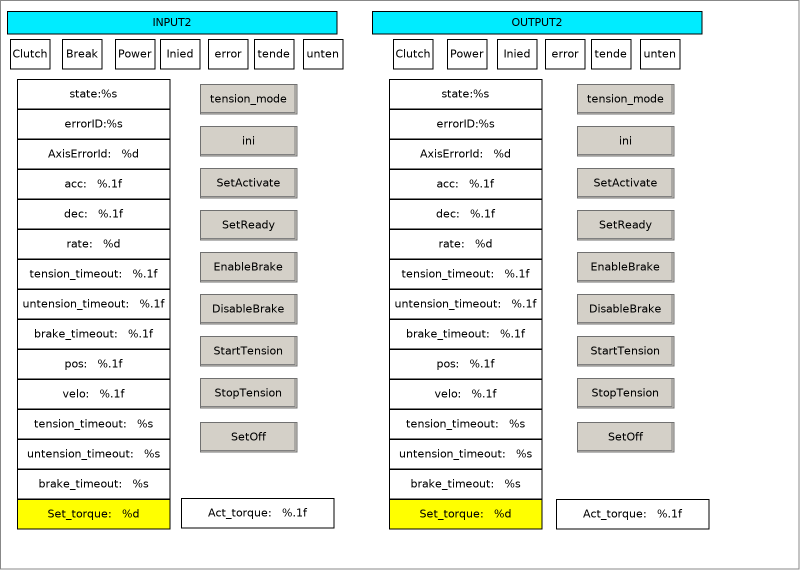
VISUALIZATION VIS_RTR_2  // 800x570
    RoundedRectangle (372,11 330x23), "OUTPUT2"
    RoundedRectangle (7,11 330x23), "INPUT2"
    Rectangle (17,79 153x30), "state:%s", colour toggle: GVL_API.stRoolToRool[3].state=100, text list: 'TextList_RTRstate', text index: GVL_API.stRoolToRool[3].state
    Rectangle (17,109 153x30), "errorID:%s", colour toggle: GVL_API.stRoolToRool[3].error_code<>0, text list: 'TextList_RTR_errorid', text index: GVL_API.stRoolToRool[3].error_code
    Rectangle (17,169 153x30), "acc: %.1f", text variable: GVL_API.stRoolToRool[3].acceleration
        OnMouseDown: write GVL_API.stRoolToRool[3].acceleration via Default
    Rectangle (17,199 153x30), "dec: %.1f", text variable: GVL_API.stRoolToRool[3].deceleration
        OnMouseDown: write GVL_API.stRoolToRool[3].deceleration via Default
    Rectangle (17,229 153x30), "rate: %d", text variable: GVL_API.stRoolToRool[3].rate
        OnMouseDown: write GVL_API.stRoolToRool[3].rate via Default
    Rectangle (17,259 153x30), "tension_timeout: %.1f", text variable: GVL_API.stRoolToRool[3].tension_timeout
        OnMouseDown: write GVL_API.stRoolToRool[3].tension_timeout via Default
    Rectangle (17,289 153x30), "untension_timeout: %.1f", text variable: GVL_API.stRoolToRool[3].untension_timeout
        OnMouseDown: write GVL_API.stRoolToRool[3].untension_timeout via Default
    Rectangle (17,319 153x30), "brake_timeout: %.1f", text variable: GVL_API.stRoolToRool[3].brake_timeout
        OnMouseDown: write GVL_API.stRoolToRool[3].brake_timeout via Default
    Rectangle (17,139 153x30), "AxisErrorId: %d", text variable: GVL_API.stRoolToRool[3].AxisErrorId
    RoundedRectangle (10,39 40x30), "Clutch", colour toggle: stOutput .bqCluthOut[3]
    RoundedRectangle (62,39 40x30), "Break", colour toggle: stOutput.bqBreakPower[3]
    Rectangle (389,79 153x30), "state:%s", colour toggle: GVL_API.stRoolToRool[4].state=100, text list: 'TextList_RTRstate', text index: GVL_API.stRoolToRool[4].state
    Rectangle (389,109 153x30), "errorID:%s", colour toggle: GVL_API.stRoolToRool[3].error_code<>0, text list: 'TextList_RTR_errorid', text index: GVL_API.stRoolToRool[4].error_code
    Rectangle (389,169 153x30), "acc: %.1f", text variable: GVL_API.stRoolToRool[4].acceleration
        OnMouseDown: write GVL_API.stRoolToRool[4].acceleration via Default
    Rectangle (389,199 153x30), "dec: %.1f", text variable: GVL_API.stRoolToRool[4].deceleration
        OnMouseDown: write GVL_API.stRoolToRool[4].deceleration via Default
    Rectangle (389,229 153x30), "rate: %d", text variable: GVL_API.stRoolToRool[4].rate
        OnMouseDown: write GVL_API.stRoolToRool[4].rate via Default
    Rectangle (389,259 153x30), "tension_timeout: %.1f", text variable: GVL_API.stRoolToRool[4].tension_timeout
        OnMouseDown: write GVL_API.stRoolToRool[4].tension_timeout via Default
    Rectangle (389,289 153x30), "untension_timeout: %.1f", text variable: GVL_API.stRoolToRool[4].untension_timeout
        OnMouseDown: write GVL_API.stRoolToRool[4].untension_timeout via Default
    Rectangle (389,319 153x30), "brake_timeout: %.1f", text variable: GVL_API.stRoolToRool[4].brake_timeout
        OnMouseDown: write GVL_API.stRoolToRool[4].brake_timeout via Default
    Rectangle (389,139 153x30), "AxisErrorId: %d", text variable: GVL_API.stRoolToRool[4].AxisErrorId
    RoundedRectangle (393,39 40x30), "Clutch", colour toggle: stOutput .bqCluthOut[4]
    Button (200,126 97x30), "ini", colour toggle: GVL_API.stRoolToRool[3].Initialize
        toggle GVL_API.stRoolToRool[3].Initialize
    Button (200,84 97x30), "tension_mode", colour toggle: GVL_API.stRoolToRool[3].tension_mode
        toggle GVL_API.stRoolToRool[3].tension_mode
    Button (200,168 97x30), "SetActivate", colour toggle: GVL_API.stRoolToRool[3].SetActivate
        toggle GVL_API.stRoolToRool[3].SetActivate
    Button (200,294 97x30), "DisableBrake", colour toggle: GVL_API.stRoolToRool[3].DisableBrake
        toggle GVL_API.stRoolToRool[3].DisableBrake
    Button (200,210 97x30), "SetReady", colour toggle: GVL_API.stRoolToRool[3].SetReady
        toggle GVL_API.stRoolToRool[3].SetReady
    Button (200,252 97x30), "EnableBrake", colour toggle: GVL_API.stRoolToRool[3].EnableBrake
        toggle GVL_API.stRoolToRool[3].EnableBrake
    Button (200,336 97x30), "StartTension", colour toggle: GVL_API.stRoolToRool[3].StartTension
        toggle GVL_API.stRoolToRool[3].StartTension
    Button (200,378 97x30), "StopTension", colour toggle: GVL_API.stRoolToRool[3].StopTension
        toggle GVL_API.stRoolToRool[3].StopTension
    Button (200,422 97x30), "SetOff", colour toggle: GVL_API.stRoolToRool[3].SetOff
        toggle GVL_API.stRoolToRool[3].SetOff
    Button (577,126 97x30), "ini", colour toggle: GVL_API.stRoolToRool[4].Initialize
        toggle GVL_API.stRoolToRool[4].Initialize
    Button (577,84 97x30), "tension_mode", colour toggle: GVL_API.stRoolToRool[4].tension_mode
        toggle GVL_API.stRoolToRool[4].tension_mode
    Button (577,168 97x30), "SetActivate", colour toggle: GVL_API.stRoolToRool[4].SetActivate
        toggle GVL_API.stRoolToRool[4].SetActivate
    Button (577,294 97x30), "DisableBrake", colour toggle: GVL_API.stRoolToRool[4].DisableBrake
        toggle GVL_API.stRoolToRool[4].DisableBrake
    Button (577,210 97x30), "SetReady", colour toggle: GVL_API.stRoolToRool[4].SetReady
        toggle GVL_API.stRoolToRool[4].SetReady
    Button (577,252 97x30), "EnableBrake", colour toggle: GVL_API.stRoolToRool[4].EnableBrake
        toggle GVL_API.stRoolToRool[4].EnableBrake
    Button (577,336 97x30), "StartTension", colour toggle: GVL_API.stRoolToRool[4].StartTension
        toggle GVL_API.stRoolToRool[4].StartTension
    Button (577,378 97x30), "StopTension", colour toggle: GVL_API.stRoolToRool[4].StopTension
        toggle GVL_API.stRoolToRool[4].StopTension
    Button (577,422 97x30), "SetOff", colour toggle: GVL_API.stRoolToRool[4].SetOff
        toggle GVL_API.stRoolToRool[4].SetOff
    RoundedRectangle (447,39 40x30), "Power", colour toggle: P_RollToRoll.FB_RoolToRool[4].REF.Status.ControlLoopClosed
    RoundedRectangle (115,39 40x30), "Power", colour toggle: P_RollToRoll.FB_RoolToRool[3].REF.Status.ControlLoopClosed
    Rectangle (17,349 153x30), "pos: %.1f", text variable: P_RollToRoll.FB_RoolToRool[3].REF.NcToPlc.ActPos
        OnMouseDown: write GVL_API.stRoolToRool[1].brake_timeout via Default
    Rectangle (17,379 153x30), "velo: %.1f", text variable: P_RollToRoll.FB_RoolToRool[3].REF.NcToPlc.ActVelo
        OnMouseDown: write GVL_API.stRoolToRool[1].brake_timeout via Default
    Rectangle (389,349 153x30), "pos: %.1f", text variable: P_RollToRoll.FB_RoolToRool[4].REF.NcToPlc.ActPos
        OnMouseDown: write GVL_API.stRoolToRool[1].brake_timeout via Default
    Rectangle (389,379 153x30), "velo: %.1f", text variable: P_RollToRoll.FB_RoolToRool[4].REF.NcToPlc.ActVelo
        OnMouseDown: write GVL_API.stRoolToRool[1].brake_timeout via Default
    Rectangle (17,409 153x30), "tension_timeout: %s", text variable: P_RollToRoll.FB_RoolToRool[3].tension_ton.ET
    Rectangle (17,439 153x30), "untension_timeout: %s", text variable: P_RollToRoll.FB_RoolToRool[3].untension_ton.ET
    Rectangle (17,469 153x30), "brake_timeout: %s", text variable: P_RollToRoll.FB_RoolToRool[3].enbreak_ton.ET
    Rectangle (389,409 153x30), "tension_timeout: %s", text variable: P_RollToRoll.FB_RoolToRool[4].tension_ton.ET
    Rectangle (389,439 153x30), "untension_timeout: %s", text variable: P_RollToRoll.FB_RoolToRool[4].untension_ton.ET
    Rectangle (389,469 153x30), "brake_timeout: %s", text variable: P_RollToRoll.FB_RoolToRool[4].enbreak_ton.ET
    Rectangle (17,499 153x30), "Set_torque: %d", text variable: HMI_RTR_set_Torque[3]
        OnMouseDown: write HMI_RTR_set_Torque[3] via Default, min 0, max 100
    Rectangle (389,499 153x30), "Set_torque: %d", text variable: HMI_RTR_set_Torque[4]
        OnMouseDown: write HMI_RTR_set_Torque[4] via Default, min 0, max 100
    Rectangle (181,498 153x30), "Act_torque: %.1f", text variable: P_RollToRoll.FB_RoolToRool[3].REF.NcToPlc.ActTorque
    Rectangle (556,499 153x30), "Act_torque: %.1f", text variable: P_RollToRoll.FB_RoolToRool[4].REF.NcToPlc.ActTorque
    RoundedRectangle (160,39 40x30), "Inied", colour toggle: P_RollToRoll.FB_RoolToRool[3].Initialized
    RoundedRectangle (208,39 40x30), "error", colour toggle: P_RollToRoll.FB_RoolToRool[3].error
    RoundedRectangle (254,39 40x30), "tende", colour toggle: P_RollToRoll.FB_RoolToRool[3].tensioned
    RoundedRectangle (303,39 40x30), "unten", colour toggle: P_RollToRoll.FB_RoolToRool[3].untensioned
    RoundedRectangle (497,39 40x30), "Inied", colour toggle: P_RollToRoll.FB_RoolToRool[4].Initialized
    RoundedRectangle (545,39 40x30), "error", colour toggle: P_RollToRoll.FB_RoolToRool[4].error
    RoundedRectangle (591,39 40x30), "tende", colour toggle: P_RollToRoll.FB_RoolToRool[4].tensioned
    RoundedRectangle (640,39 40x30), "unten", colour toggle: P_RollToRoll.FB_RoolToRool[4].untensioned
END_VISUALIZATION

(* stored: Version 1.1.0.1, ProductVersion 3.1.4024.11
   Visu VIS_RTR_2: Id {a9e25b22-1328-45e3-ac25-7d7471d9655a} *)
